{attribute 'OPC.UA.DA' := '1'}
TYPE ST_Binder :
STRUCT
	State		:	ST_BinderState;		// State of the Binder
	FromBinder	:	ST_FromBinder;		// Data Recevied from the Binder
	ToBinder	:	ST_ToBinder;		// Data Sent to the Binder
END_STRUCT
END_TYPE

(* stored: Version 1.1.0.1, ProductVersion 3.1.4024.6
   DUT ST_Binder: Id {1914bf23-7c15-4bb4-872a-03f65b6603e9} *)
